// TIA Portal V15.1 export
// export: Created 2026-01-15T16:29:42.237043Z, ExportSetting WithDefaults, WithReadOnly, DisplayName Totally Integrated Automation Portal, DisplayVersion V15.1 Update 8, DisplayName TIA Portal Openness, DisplayVersion V15.1 Update 8, DisplayName STEP 7 Professional, DisplayVersion V15.1 Update 8, DisplayName WinCC Advanced, DisplayVersion V15.1 Update 8
FUNCTION "5. QUA TRINH NAP LIEU" : Void   // FC5, LAD
{ S7_Optimized_Access := 'TRUE' }
VERSION : 0.1
// stored: AutoNumber true, CodeModifiedDate 2026-01-15T16:25:52.514227Z, CompileDate 2026-01-15T16:25:52.5840608Z, CreationDate 2026-01-15T16:22:49.8270549Z, HandleErrorsWithinBlock false, InterfaceModifiedDate 2023-12-12T15:54:48.677177Z, IsConsistent true, IsIECCheckEnabled false, IsKnowHowProtected false, IsWriteProtected false, LibraryConformanceStatus Warning: The object contains access to global data blocks. Warning: The block contains direct access to inputs, outputs, bit memories, indirect access to the registry or indirect access to external memory areas that are unknown at the time of compilation., ModifiedDate 2026-01-15T16:25:52.514227Z, ParameterModified 2023-12-12T15:54:48.677177Z, PLCSimAdvancedSupport false, SetENOAutomatically False, StructureModified 2023-12-12T15:54:48.677177Z, UDAEnableTagReadback false
   VAR_OUTPUT
      XA_PTG : Bool;
      XA_CEM1 : Bool;
      XA_CEM2 : Bool;
      XA_WAT1 : Bool;
      XA_WAT2 : Bool;
      XA_ADD1 : Bool;
      XA_ADD2 : Bool;
   END_VAR
BEGIN

REGION Network 1: Van xả phễu chờ
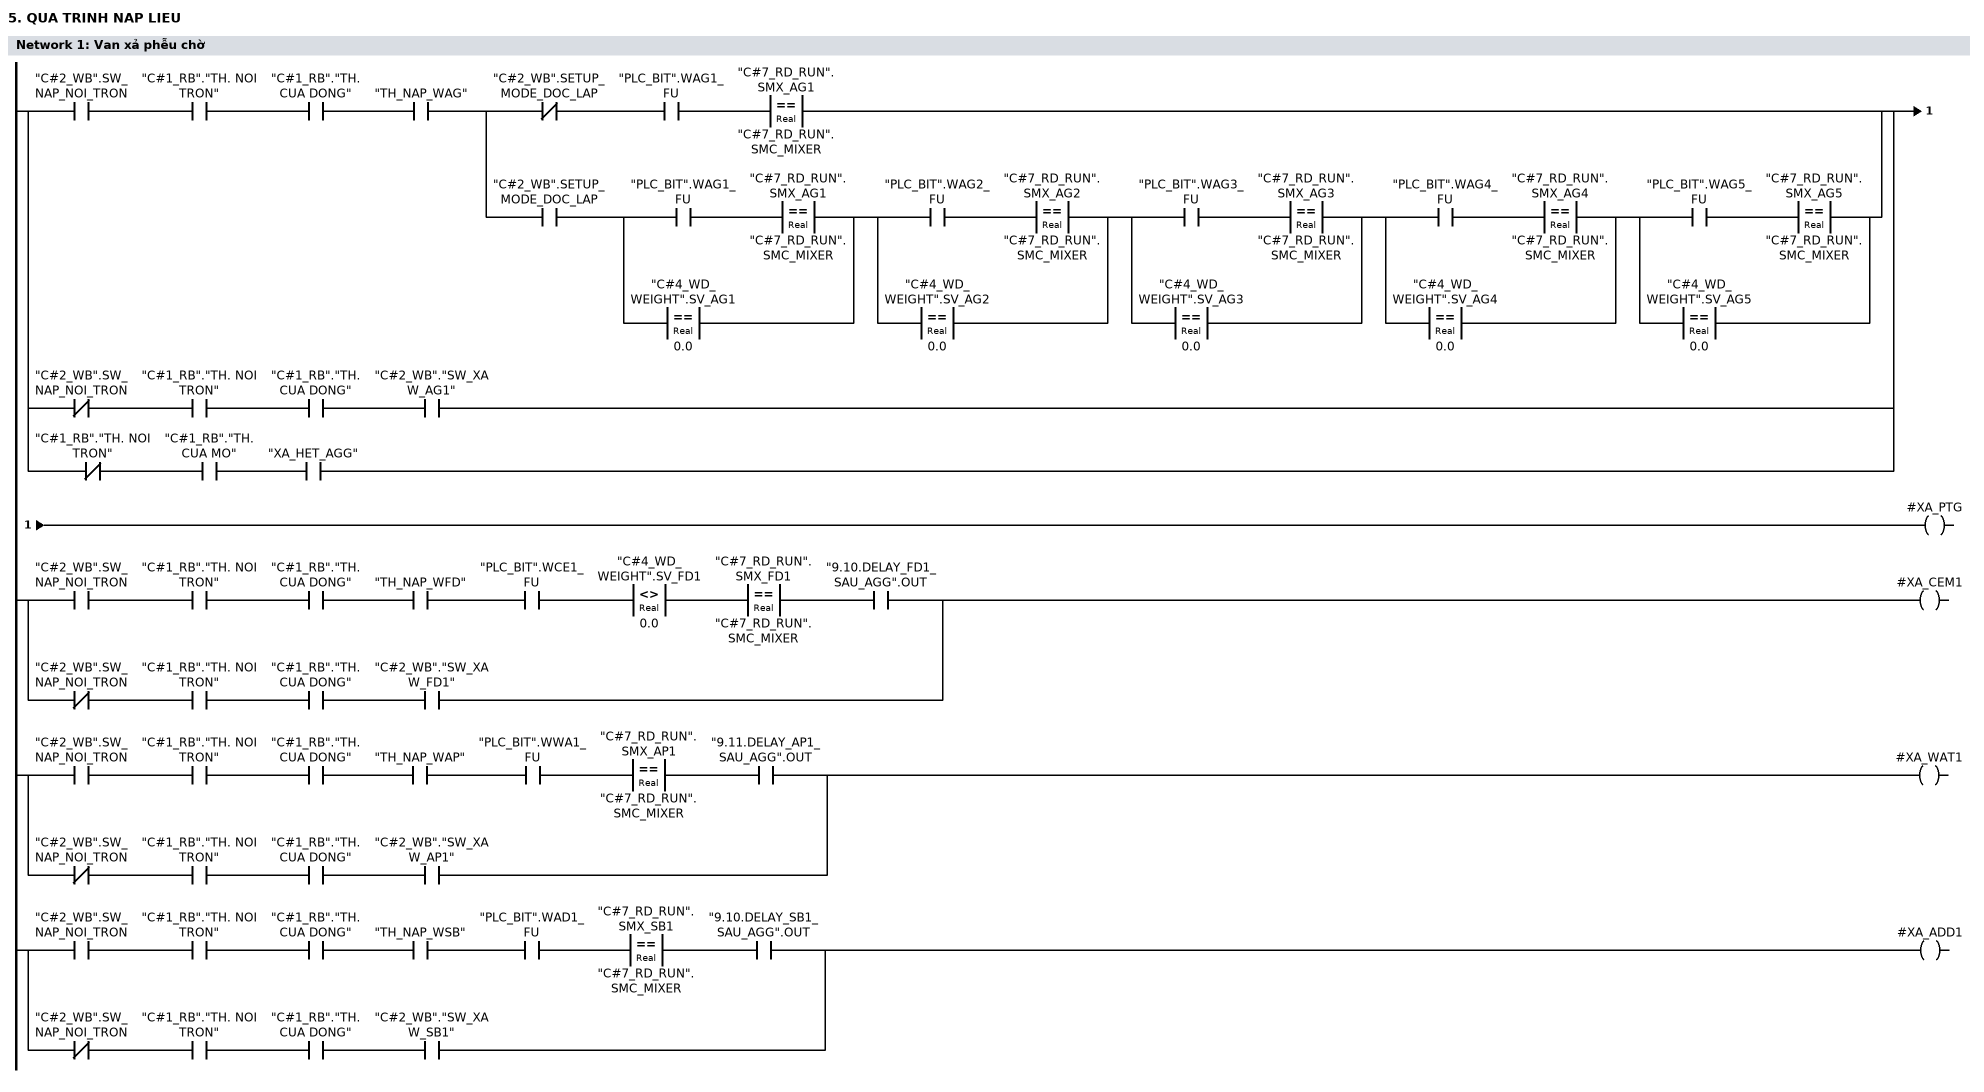
   RUNG wire#powerrail
      Contact( "C#2_WB".SW_NAP_NOI_TRON )
      Contact( "C#1_RB"."TH. NOI TRON" )
      Contact( "C#1_RB"."TH. CUA DONG" )
      Contact( "TH_NAP_WAG" )
      wire#w1
      I_Contact( "C#2_WB".SETUP_MODE_DOC_LAP )
      Contact( "PLC_BIT".WAG1_FU )
      { S7_Templates := "SrcType := Real" } EQ_Contact(in1 := "C#7_RD_RUN".SMX_AG1, in2 := "C#7_RD_RUN".SMC_MIXER)
      wire#w2
      Coil( #XA_PTG )
   END_RUNG
   RUNG wire#w1
      Contact( "C#2_WB".SETUP_MODE_DOC_LAP )
      wire#w3
      Contact( "PLC_BIT".WAG1_FU )
      { S7_Templates := "SrcType := Real" } EQ_Contact(in1 := "C#7_RD_RUN".SMX_AG1, in2 := "C#7_RD_RUN".SMC_MIXER)
      wire#w4
      Contact( "PLC_BIT".WAG2_FU )
      { S7_Templates := "SrcType := Real" } EQ_Contact(in1 := "C#7_RD_RUN".SMX_AG2, in2 := "C#7_RD_RUN".SMC_MIXER)
      wire#w5
      Contact( "PLC_BIT".WAG3_FU )
      { S7_Templates := "SrcType := Real" } EQ_Contact(in1 := "C#7_RD_RUN".SMX_AG3, in2 := "C#7_RD_RUN".SMC_MIXER)
      wire#w6
      Contact( "PLC_BIT".WAG4_FU )
      { S7_Templates := "SrcType := Real" } EQ_Contact(in1 := "C#7_RD_RUN".SMX_AG4, in2 := "C#7_RD_RUN".SMC_MIXER)
      wire#w7
      Contact( "PLC_BIT".WAG5_FU )
      { S7_Templates := "SrcType := Real" } EQ_Contact(in1 := "C#7_RD_RUN".SMX_AG5, in2 := "C#7_RD_RUN".SMC_MIXER)
   END_RUNG wire#w2
   RUNG wire#w3
      { S7_Templates := "SrcType := Real" } EQ_Contact(in1 := "C#4_WD_WEIGHT".SV_AG1, in2 := 0.0)
   END_RUNG wire#w4
   RUNG wire#w4
      { S7_Templates := "SrcType := Real" } EQ_Contact(in1 := "C#4_WD_WEIGHT".SV_AG2, in2 := 0.0)
   END_RUNG wire#w5
   RUNG wire#w5
      { S7_Templates := "SrcType := Real" } EQ_Contact(in1 := "C#4_WD_WEIGHT".SV_AG3, in2 := 0.0)
   END_RUNG wire#w6
   RUNG wire#w6
      { S7_Templates := "SrcType := Real" } EQ_Contact(in1 := "C#4_WD_WEIGHT".SV_AG4, in2 := 0.0)
   END_RUNG wire#w7
   RUNG wire#w7
      { S7_Templates := "SrcType := Real" } EQ_Contact(in1 := "C#4_WD_WEIGHT".SV_AG5, in2 := 0.0)
   END_RUNG wire#w2
   RUNG wire#powerrail
      I_Contact( "C#2_WB".SW_NAP_NOI_TRON )
      Contact( "C#1_RB"."TH. NOI TRON" )
      Contact( "C#1_RB"."TH. CUA DONG" )
      Contact( "C#2_WB"."SW_XA W_AG1" )
   END_RUNG wire#w2
   RUNG wire#powerrail
      I_Contact( "C#1_RB"."TH. NOI TRON" )
      Contact( "C#1_RB"."TH. CUA MO" )
      Contact( "XA_HET_AGG" )
   END_RUNG wire#w2
   RUNG wire#powerrail
      Contact( "C#2_WB".SW_NAP_NOI_TRON )
      Contact( "C#1_RB"."TH. NOI TRON" )
      Contact( "C#1_RB"."TH. CUA DONG" )
      Contact( "TH_NAP_WFD" )
      Contact( "PLC_BIT".WCE1_FU )
      { S7_Templates := "SrcType := Real" } NE_Contact(in1 := "C#4_WD_WEIGHT".SV_FD1, in2 := 0.0)
      { S7_Templates := "SrcType := Real" } EQ_Contact(in1 := "C#7_RD_RUN".SMX_FD1, in2 := "C#7_RD_RUN".SMC_MIXER)
      Contact( "9.10.DELAY_FD1_SAU_AGG".OUT )
      wire#w8
      Coil( #XA_CEM1 )
   END_RUNG
   RUNG wire#powerrail
      I_Contact( "C#2_WB".SW_NAP_NOI_TRON )
      Contact( "C#1_RB"."TH. NOI TRON" )
      Contact( "C#1_RB"."TH. CUA DONG" )
      Contact( "C#2_WB"."SW_XA W_FD1" )
   END_RUNG wire#w8
   RUNG wire#powerrail
      Contact( "C#2_WB".SW_NAP_NOI_TRON )
      Contact( "C#1_RB"."TH. NOI TRON" )
      Contact( "C#1_RB"."TH. CUA DONG" )
      Contact( "TH_NAP_WAP" )
      Contact( "PLC_BIT".WWA1_FU )
      { S7_Templates := "SrcType := Real" } EQ_Contact(in1 := "C#7_RD_RUN".SMX_AP1, in2 := "C#7_RD_RUN".SMC_MIXER)
      Contact( "9.11.DELAY_AP1_SAU_AGG".OUT )
      wire#w9
      Coil( #XA_WAT1 )
   END_RUNG
   RUNG wire#powerrail
      I_Contact( "C#2_WB".SW_NAP_NOI_TRON )
      Contact( "C#1_RB"."TH. NOI TRON" )
      Contact( "C#1_RB"."TH. CUA DONG" )
      Contact( "C#2_WB"."SW_XA W_AP1" )
   END_RUNG wire#w9
   RUNG wire#powerrail
      Contact( "C#2_WB".SW_NAP_NOI_TRON )
      Contact( "C#1_RB"."TH. NOI TRON" )
      Contact( "C#1_RB"."TH. CUA DONG" )
      Contact( "TH_NAP_WSB" )
      Contact( "PLC_BIT".WAD1_FU )
      { S7_Templates := "SrcType := Real" } EQ_Contact(in1 := "C#7_RD_RUN".SMX_SB1, in2 := "C#7_RD_RUN".SMC_MIXER)
      Contact( "9.10.DELAY_SB1_SAU_AGG".OUT )
      wire#w10
      Coil( #XA_ADD1 )
   END_RUNG
   RUNG wire#powerrail
      I_Contact( "C#2_WB".SW_NAP_NOI_TRON )
      Contact( "C#1_RB"."TH. NOI TRON" )
      Contact( "C#1_RB"."TH. CUA DONG" )
      Contact( "C#2_WB"."SW_XA W_SB1" )
   END_RUNG wire#w10
   // the same network as SCL:
   #XA_PTG := ("C#2_WB".SW_NAP_NOI_TRON AND "C#1_RB"."TH. NOI TRON" AND "C#1_RB"."TH. CUA DONG" AND "TH_NAP_WAG" AND ((NOT "C#2_WB".SETUP_MODE_DOC_LAP AND "PLC_BIT".WAG1_FU AND ("C#7_RD_RUN".SMX_AG1 = "C#7_RD_RUN".SMC_MIXER)) OR ("C#2_WB".SETUP_MODE_DOC_LAP AND (("PLC_BIT".WAG1_FU AND ("C#7_RD_RUN".SMX_AG1 = "C#7_RD_RUN".SMC_MIXER)) OR ("C#4_WD_WEIGHT".SV_AG1 = 0.0)) AND (("PLC_BIT".WAG2_FU AND ("C#7_RD_RUN".SMX_AG2 = "C#7_RD_RUN".SMC_MIXER)) OR ("C#4_WD_WEIGHT".SV_AG2 = 0.0)) AND (("PLC_BIT".WAG3_FU AND ("C#7_RD_RUN".SMX_AG3 = "C#7_RD_RUN".SMC_MIXER)) OR ("C#4_WD_WEIGHT".SV_AG3 = 0.0)) AND (("PLC_BIT".WAG4_FU AND ("C#7_RD_RUN".SMX_AG4 = "C#7_RD_RUN".SMC_MIXER)) OR ("C#4_WD_WEIGHT".SV_AG4 = 0.0)) AND (("PLC_BIT".WAG5_FU AND ("C#7_RD_RUN".SMX_AG5 = "C#7_RD_RUN".SMC_MIXER)) OR ("C#4_WD_WEIGHT".SV_AG5 = 0.0))))) OR (NOT "C#2_WB".SW_NAP_NOI_TRON AND "C#1_RB"."TH. NOI TRON" AND "C#1_RB"."TH. CUA DONG" AND "C#2_WB"."SW_XA W_AG1") OR (NOT "C#1_RB"."TH. NOI TRON" AND "C#1_RB"."TH. CUA MO" AND "XA_HET_AGG");
   #XA_CEM1 := ("C#2_WB".SW_NAP_NOI_TRON AND "C#1_RB"."TH. NOI TRON" AND "C#1_RB"."TH. CUA DONG" AND "TH_NAP_WFD" AND "PLC_BIT".WCE1_FU AND ("C#4_WD_WEIGHT".SV_FD1 <> 0.0) AND ("C#7_RD_RUN".SMX_FD1 = "C#7_RD_RUN".SMC_MIXER) AND "9.10.DELAY_FD1_SAU_AGG".OUT) OR (NOT "C#2_WB".SW_NAP_NOI_TRON AND "C#1_RB"."TH. NOI TRON" AND "C#1_RB"."TH. CUA DONG" AND "C#2_WB"."SW_XA W_FD1");
   #XA_WAT1 := ("C#2_WB".SW_NAP_NOI_TRON AND "C#1_RB"."TH. NOI TRON" AND "C#1_RB"."TH. CUA DONG" AND "TH_NAP_WAP" AND "PLC_BIT".WWA1_FU AND ("C#7_RD_RUN".SMX_AP1 = "C#7_RD_RUN".SMC_MIXER) AND "9.11.DELAY_AP1_SAU_AGG".OUT) OR (NOT "C#2_WB".SW_NAP_NOI_TRON AND "C#1_RB"."TH. NOI TRON" AND "C#1_RB"."TH. CUA DONG" AND "C#2_WB"."SW_XA W_AP1");
   #XA_ADD1 := ("C#2_WB".SW_NAP_NOI_TRON AND "C#1_RB"."TH. NOI TRON" AND "C#1_RB"."TH. CUA DONG" AND "TH_NAP_WSB" AND "PLC_BIT".WAD1_FU AND ("C#7_RD_RUN".SMX_SB1 = "C#7_RD_RUN".SMC_MIXER) AND "9.10.DELAY_SB1_SAU_AGG".OUT) OR (NOT "C#2_WB".SW_NAP_NOI_TRON AND "C#1_RB"."TH. NOI TRON" AND "C#1_RB"."TH. CUA DONG" AND "C#2_WB"."SW_XA W_SB1");
END_REGION
END_FUNCTION
